(* LS Electric XG5000 project: 241007_사용자정의펑션 *)
(* PLC LSPLC *)

FUNCTION 시간검출 : ARRAY[0..5] OF WORD
VAR_INPUT
    _RTC_TIME_0 : BYTE; (* _RTC_TIME[0] *)
    _RTC_TIME_1 : BYTE;
    _RTC_TIME_2 : BYTE;
    _RTC_TIME_3 : BYTE;
    _RTC_TIME_4 : BYTE;
    _RTC_TIME_5 : BYTE;
END_VAR

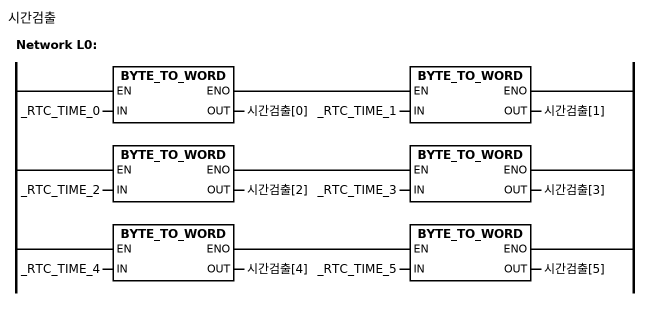
(* Rung L0 *)
시간검출[0] := BYTE_TO_WORD(_RTC_TIME_0);
시간검출[1] := BYTE_TO_WORD(_RTC_TIME_1);
시간검출[2] := BYTE_TO_WORD(_RTC_TIME_2);
시간검출[3] := BYTE_TO_WORD(_RTC_TIME_3);
시간검출[4] := BYTE_TO_WORD(_RTC_TIME_4);
시간검출[5] := BYTE_TO_WORD(_RTC_TIME_5);
END_FUNCTION

PROGRAM NewProgram (* task: 스캔 프로그램 *)
VAR
    트리거 AT %IX0.0.0 : BOOL;
    현재시간 : ARRAY[0..5] OF WORD;
END_VAR

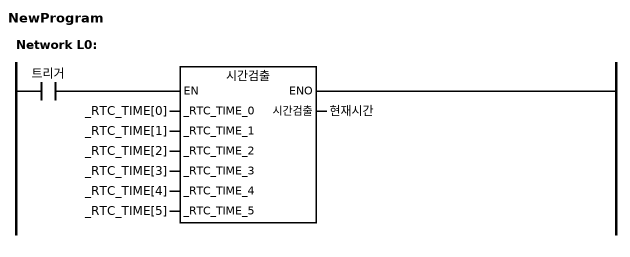
(* Rung L0 *)
IF 트리거 THEN
    현재시간 := 시간검출(_RTC_TIME_0 := _RTC_TIME[0], _RTC_TIME_1 := _RTC_TIME[1], _RTC_TIME_2 := _RTC_TIME[2], _RTC_TIME_3 := _RTC_TIME[3], _RTC_TIME_4 := _RTC_TIME[4], _RTC_TIME_5 := _RTC_TIME[5]);
END_IF;
END_PROGRAM